// ==============================================================================
// FC_Route_Supervisor - Супервізор маршрутів (Mailbox Pattern v3.1)
// ==============================================================================
// Версія: 3.2.2
// Дата: 2026-03-01
// ==============================================================================

FUNCTION "FC_Route_Supervisor" : VOID
{ S7_Optimized_Access := 'TRUE' }
VERSION : 3.1



VAR_TEMP
  i                : USINT;
  commitIn         : UDINT;
  commitAck        : UDINT;
  routeId          : USINT;
  currentState     : UINT;
  isActive         : BOOL;
  isStoppable      : BOOL;   // STARTING OR RUNNING OR STOPPING (не VALIDATING)
  cmdAllowed       : BOOL;
  processedRouteId : USINT;
  pendingWarning   : USINT;
  savedWarnings    : ARRAY[1.."ROUTES_COUNT"] OF USINT;  // Зберегти RS_Warning
  j                : INT;                                // ітератор кроків у Cleanup
  stepBound        : INT;                                // верхня межа циклу (≤ROUTE_MAX_STEPS-1)
  innerSlot        : UINT;                               // слот механізму у Cleanup
  routeAllReleased : BOOL;                               // чи всі механізми звільнені
END_VAR

BEGIN

    // Ініціалізація
    processedRouteId := 0;
    pendingWarning := "RS_WARNING_OK";

    // =========================================================
    // 1. ЗБЕРЕГТИ RS_Warning перед FSM
    // =========================================================
    // ✅ КРИТИЧНО: FSM затирає RS_Warning кожного циклу
    FOR i := 1 TO "ROUTES_COUNT" DO
        savedWarnings[i] := "DB_PlcToScada_RouteStatus".RoutesSts[i].RS_Warning;
    END_FOR;

    // =========================================================
    // 2. MAILBOX: Детект нової команди
    // =========================================================
    commitIn  := "DB_ScadaToPlc_RouteCmd".HDR_Commit;
    commitAck := "DB_PlcToScada_RouteStatus".ACK_CommitApplied;

    IF commitIn <> commitAck THEN

        // =========================================================
        // 3. MAILBOX: Валідація RouteId
        // =========================================================
        routeId := "DB_ScadaToPlc_RouteCmd".HDR_RouteId;

        // Невалідний RouteId → ACK (mailbox не блокується) + RETURN
        IF (routeId < 1) OR (routeId > "ROUTES_COUNT") THEN
            "DB_PlcToScada_RouteStatus".ACK_CommitApplied := commitIn;
            "DB_PlcToScada_RouteStatus".ACK_RouteId := 0;
            RETURN;
        END_IF;

        // =========================================================
        // 4. MAILBOX: Перевірка стану маршруту
        // =========================================================
        currentState := "DB_PlcToScada_RouteStatus".RoutesSts[routeId].RS_State;

        isActive := (currentState = "ROUTE_STS_VALIDATING") OR
                    (currentState = "ROUTE_STS_STARTING") OR
                    (currentState = "ROUTE_STS_RUNNING") OR
                    (currentState = "ROUTE_STS_STOPPING");

        // STOP_OP дозволено тільки з STARTING/RUNNING/STOPPING
        // У VALIDATING механізми ще не захоплені → STOP_OP беззмістовний
        isStoppable := (currentState = "ROUTE_STS_STARTING") OR
                       (currentState = "ROUTE_STS_RUNNING")  OR
                       (currentState = "ROUTE_STS_STOPPING");

        cmdAllowed := FALSE;

        // Перевірка дозволеності команди
        IF "DB_ScadaToPlc_RouteCmd".CMD_Route.RC_Cmd = "RT_CMD_START" THEN
            IF isActive THEN
                // START для активного → ігнорувати з попередженням
                pendingWarning := "RS_WARNING_IGNORED_CMD";
                cmdAllowed := FALSE;
            ELSE
                // START для неактивного → дозволено
                pendingWarning := "RS_WARNING_OK";
                cmdAllowed := TRUE;
            END_IF;

        ELSIF "DB_ScadaToPlc_RouteCmd".CMD_Route.RC_Cmd = "RT_CMD_STOP_OP" THEN
            IF isStoppable THEN
                // STOP_OP для STARTING/RUNNING/STOPPING — дозволено
                pendingWarning := "RS_WARNING_OK";
                cmdAllowed := TRUE;
            ELSE
                // STOP_OP для VALIDATING/IDLE/REJECTED/ABORTED — ігнорувати з попередженням
                pendingWarning := "RS_WARNING_IGNORED_CMD";
                cmdAllowed := FALSE;
            END_IF;

        ELSE
            // RT_CMD_NONE або невідома команда
            cmdAllowed := FALSE;
        END_IF;

        // =========================================================
        // 5. MAILBOX: Копіювання команди у RouteExecutor
        // =========================================================
        IF cmdAllowed THEN
            "DB_Plc_RouteExecutor".Routes[routeId] := "DB_ScadaToPlc_RouteCmd".CMD_Route;
        END_IF;

        // =========================================================
        // 6. MAILBOX: Підтвердження (ACK)
        // =========================================================
        "DB_PlcToScada_RouteStatus".ACK_CommitApplied := commitIn;
        "DB_PlcToScada_RouteStatus".ACK_RouteId := routeId;

        // Запам'ятати який маршрут обробили
        processedRouteId := routeId;

    END_IF;

    // =========================================================
    // 7. FSM: Виконання всіх маршрутів
    // =========================================================
    FOR i := 1 TO "ROUTES_COUNT" DO

        "FC_RouteFSM"(
            RouteIdx          := INT_TO_USINT(i),
            Cmd               := "DB_Plc_RouteExecutor".Routes[i],
            Mechs             := "DB_Mechs".Mechs,
            Fsm               := "DB_Plc_RouteFsm".RoutesFsm[i],
            Sts               => "DB_PlcToScada_RouteStatus".RoutesSts[i]
        );

    END_FOR;

    // =========================================================
    // 8. ✅ ВІДНОВИТИ RS_Warning після FSM
    // =========================================================
    FOR i := 1 TO "ROUTES_COUNT" DO
        IF i = processedRouteId THEN
            // Для обробленого маршруту → встановити новий Warning
            "DB_PlcToScada_RouteStatus".RoutesSts[i].RS_Warning := pendingWarning;
        ELSE
            // Для інших маршрутів → відновити збережений Warning
            "DB_PlcToScada_RouteStatus".RoutesSts[i].RS_Warning := savedWarnings[i];
        END_IF;
    END_FOR;

    // =========================================================
    // 9. CLEANUP: Очищення RouteExecutor після завершення
    // =========================================================
    FOR i := 1 TO "ROUTES_COUNT" DO
        // Пропустити маршрут, який щойно отримав нову команду
        IF i = processedRouteId THEN
            CONTINUE;
        END_IF;

        currentState := "DB_PlcToScada_RouteStatus".RoutesSts[i].RS_State;

        // Очищати маршрути у фінальних станах (REJECTED включено — без цього FSM застряє)
        IF (currentState = "ROUTE_STS_ABORTED") OR (currentState = "ROUTE_STS_IDLE")
        OR (currentState = "ROUTE_STS_REJECTED") THEN

            // Перевірити чи є ще механізми що належать цьому маршруту.
            //
            // Якщо є — НЕ очищати RC_StepCount. Це зберігає список слотів живим для:
            //   - GlobalSafetyStop block: ретраює CMD_RELEASE_OWNER кожен цикл
            //     (поки GlobalSafetyStop активний і safetyHit = TRUE блокує FSM)
            //   - FSM ABORTED retry: ретраює коли safetyHit = FALSE
            //   Обидва варіанти завершаться успішно коли механізм досягне STS_IDLE/FAULT.
            //
            // Після того як всі механізми звільнені → Cleanup нулює → FSM → IDLE.
            //
            // Захист: innerSlot > MECHS_COUNT → пропускаємо (невалідний слот не читаємо).
            routeAllReleased := TRUE;
            stepBound := USINT_TO_INT("DB_Plc_RouteExecutor".Routes[i].RC_StepCount);
            IF stepBound > "ROUTE_MAX_STEPS" THEN stepBound := "ROUTE_MAX_STEPS"; END_IF;
            FOR j := 1 TO stepBound DO
                innerSlot := "DB_Plc_RouteExecutor".Routes[i].RC_Steps[j].RS_Slot;
                IF innerSlot <= "MECHS_COUNT" THEN
                    IF ("DB_Mechs".Mechs[innerSlot].OwnerCur   = "OWNER_ROUTE") AND
                       ("DB_Mechs".Mechs[innerSlot].OwnerCurId = INT_TO_UINT(i)) THEN
                        routeAllReleased := FALSE;
                        EXIT;
                    END_IF;
                END_IF;
            END_FOR;

            IF routeAllReleased THEN
                "DB_Plc_RouteExecutor".Routes[i].RC_Cmd       := "RT_CMD_NONE";
                "DB_Plc_RouteExecutor".Routes[i].RC_StepCount := 0;
            END_IF;

        END_IF;
    END_FOR;

END_FUNCTION
